// TwinCAT 3 PLC project PLC1
// ProgramVersion: 3.1.4026.25
// libraries:
//   Tc2_EtherCAT, * (Beckhoff Automation GmbH)
//   Tc2_MC2, * (Beckhoff Automation GmbH)
//   Tc2_Standard, * (Beckhoff Automation GmbH)
//   Tc2_System, * (Beckhoff Automation GmbH)
// project tree:
//   DUTs/ ST_DISDiagnosisMX.TcDUT, ST_DISInputsMX.TcDUT, ST_DOSDiagnosisMX.TcDUT, ST_DOSOutputsMX.TcDUT, ST_EFUInputsMX.TcDUT, ST_EFUOutputsMX.TcDUT, ST_IoModulMO1008.TcDUT, ST_IoModulMO2008.TcDUT, ST_IoModulMO2338.TcDUT, ST_MS4208.TcDUT, ST_PSUInputsMX.TcDUT
//   / PlcTask.TcTTO
//   POUs/ FB_RunOutputs.TcPOU, MAIN.TcPOU
// real-time tasks:
//   TASK PlcTask: cycle T#10ms, priority 20, ADS port 350
// motion (NC):
//   TASK NC-Task 1 SAF: cycle T#2ms, priority 4, ADS port 501
//   TASK NC-Task 1 SVB: cycle T#10ms, priority 8, ADS port 511
//   AXIS Axis 1 (id 1)
//     Dynamic: Acceleration=547.653, Deceleration=547.653, Jerk=1642.959
//     Velo: RefSearch=3.65102, RefSync=3.65102, SlowManual=12.5, FastManual=75, Fast=365.102, Maximum=365.102
//     OtherSettings: AllowMotionCmdToSlave=true
//     encoder EncType=19
//       EncPara: ScaleFactorNumerator=5, ScaleFactorDenominator=1048576, MaxCount=#xffffffff
//     drive DrvType=16
//       DrvPara: MaxCount=#xffffffff, DriveControlDWord=#x00020100
//         Analog: VeloReferenz=401.6122, VeloScale=32, TorqueSetpointScale=10, ScaleFactorActTorque=0.1
//         TimeComp: TaskDelayCycles=1
//     controller CtrType=1
//       CtrPara: PriorControlFactor=1
//         Observer: BandWidth=20
// I/O:
//   DEVICE Device 1 (EtherCAT), AmsNetId 192.168.7.189.2.1
//     Term 1 (MB1200-0000) [MB1200-0000 MX EtherCAT infeed]
//       Term 2 (MB1100-0002) [MB1100-0002 (Bluetooth gateway)]
//         Term 3 (MX Occupied Slot) [MX occupied Slot]
//         Term 4 (MX Occupied Slot) [MX occupied Slot]
//         Term 5 (MX Occupied Slot) [MX occupied Slot]
//         Term 6 (MS1010-1002-1334) [MS1010-1002-1334 Power infeed + forwarding, 230 V AC/10 A, 24 V DC/7A power supply, B17]
//         Term 7 (MO7221-0000-1114) [MO7221-0000-1114 1-channel motion interface, servomotor, 24 V DC/8 A, OCT, B17]
//           startup 32785:21 := 0E01 // DRV Motor Settings Ch.1 / Commutation offset
//           startup 32785:27 := E02E0000 // DRV Motor Settings Ch.1 / Motor speed limitation
//           startup 28688:3 := 08 // DRV Outputs Ch.1 / Modes of operation
//           startup 28688:16 := FF7F // DRV Outputs Ch.1 / Positive torque limit value
//           startup 28688:17 := FF7F // DRV Outputs Ch.1 / Negative torque limit value
//           startup 32784:87 := 64 // DRV Amplifier Settings Ch.1 / Position loop velocity feed forward gain
//           startup 32784:109 := 64000000 // DRV Amplifier Settings Ch.1 / Torque feed forward gain
//           startup 28688:11 := D007 // DRV Outputs Ch.1 / Torque limitation
//           startup 32784:19 := 9B00 // DRV Amplifier Settings Ch.1 / Current loop proportional gain
//           startup 32784:18 := 1200 // DRV Amplifier Settings Ch.1 / Current loop integral time
//           startup 32784:21 := C5000000 // DRV Amplifier Settings Ch.1 / Velocity loop proportional gain
//           startup 32784:20 := 96000000 // DRV Amplifier Settings Ch.1 / Velocity loop integral time
//         Term 8 (MB1120-0000) [MB1120 backplane junction]
//           Term 9 (MS4208-2003-1112) [MS4208-2003-1112 EtherCAT power output, EtherCAT, 24 V DC, 8 A, M12, switchable]
//             Term 24 (EK1100) [EK1100 EtherCAT Coupler (2A E-Bus)]
//               Term 25 (ED1008) [ED1008 | 8-ch. dig. input, 24 V DC, 3 ms, push-in]
//               Term 26 (ED2008) [ED2008 | 8-ch. dig. output, 24 V DC, 0.5 A, push-in]
//               Term 31 (ED4078) [ED4078 | 8-ch. ana. output, multi-function, ±10 V, ±20 mA, 16 bit, single-ended, 2 ksps, push-in]
//               Term 27 (ED5112) [ED5112 | 2-ch. encoder interface, incremental, 5 V DC (DIFF RS422, TTL, open collector), 5 MHz, push-in, 2 x AB/1 x ABC]
//               Term 32 (EL9011) [EL9011 End Terminal]
//         Term 10 (MO1008-0000-1111) [MO1008-0000-1111 8 Ch. Dig. Input 24V, M8]
//         Term 11 (MO2008-0000-1111) [MO2008-0000-1111 8 Ch. Dig. Output 24V, M8]
//         Term 12 (MO2338-0000-1112) [MO2338-0000-1112 8 Ch. digital combi 24V 0.5A, M12]
//         Term 15 (EL9011) [EL9011 End Terminal]
//       Term 13 (MS1110-0000) [MS1110-0000 | System module, EtherCAT extension]
// variable links:
//   NC-Task 1 SAF/Axes/Axis 1 <-> Device 1 (EtherCAT)/Term 1 (MB1200-0000)/Term 2 (MB1100-0002)/Term 7 (MO7221-0000-1114)
//     Drive/Inputs/In/nDataIn1 <-> DRV Following error actual value/Following error actual value
//     Drive/Inputs/In/nDataIn3[0] <-> DRV Torque actual value/Torque actual value
//     Drive/Inputs/In/nDcOutputTime <-> InfoData/DcOutputShift
//     Drive/Inputs/In/nState1 <-> DRV Statusword/Statusword
//     Drive/Inputs/In/nState2 <-> DRV Statusword/Statusword @bit 8
//     Drive/Inputs/In/nState4 @bit 1 <-> WcState/InputToggle
//     Drive/Inputs/In/nState4 <-> WcState/WcState
//     Drive/Outputs/Out/nCtrl1 <-> DRV Controlword/Controlword
//     Drive/Outputs/Out/nCtrl2 <-> DRV Controlword/Controlword @bit 8
//     Drive/Outputs/Out/nDataOut1 <-> DRV Target position/Target position
//     Enc/Inputs/In/nDataIn1 <-> FB Position/Position
//     Enc/Inputs/In/nDcInputTime <-> InfoData/DcInputShift
//     Enc/Inputs/In/nState4 @bit 1 <-> WcState/InputToggle
//     Enc/Inputs/In/nState4 <-> WcState/WcState
//   PLC1/PLC1 Instance <-> Device 1 (EtherCAT)
//     PlcTask Inputs/MAIN.nConfiguredSlaveCount <-> InfoData/CfgSlaveCount
//     PlcTask Inputs/MAIN.stAMSNetID <-> InfoData/AmsNetId
//   PLC1/PLC1 Instance <-> Device 1 (EtherCAT)/Term 1 (MB1200-0000)/Term 2 (MB1100-0002)
//     PlcTask Outputs/MAIN.bActivatePairingMode <-> BTG Outputs/Control/Activate Pairing
//     PlcTask Outputs/MAIN.bEnableBluetoothDiagnosis <-> BTG Outputs/Control/Enable Bluetooth
//   PLC1/PLC1 Instance <-> Device 1 (EtherCAT)/Term 1 (MB1200-0000)/Term 2 (MB1100-0002)/Term 10 (MO1008-0000-1111)
//     PlcTask Inputs/MAIN.stIoModulSlot8.stDISDiagnosis.bWirebreakCh1 <-> DIP Diagnosis/Wirebreak Ch1 X01-4
//     PlcTask Inputs/MAIN.stIoModulSlot8.stDISDiagnosis.bWirebreakCh2 <-> DIP Diagnosis/Wirebreak Ch2 X02-4
//     PlcTask Inputs/MAIN.stIoModulSlot8.stDISDiagnosis.bWirebreakCh3 <-> DIP Diagnosis/Wirebreak Ch3 X03-4
//     PlcTask Inputs/MAIN.stIoModulSlot8.stDISDiagnosis.bWirebreakCh4 <-> DIP Diagnosis/Wirebreak Ch4 X04-4
//     PlcTask Inputs/MAIN.stIoModulSlot8.stDISDiagnosis.bWirebreakCh5 <-> DIP Diagnosis/Wirebreak Ch5 X05-4
//     PlcTask Inputs/MAIN.stIoModulSlot8.stDISDiagnosis.bWirebreakCh6 <-> DIP Diagnosis/Wirebreak Ch6 X06-4
//     PlcTask Inputs/MAIN.stIoModulSlot8.stDISDiagnosis.bWirebreakCh7 <-> DIP Diagnosis/Wirebreak Ch7 X07-4
//     PlcTask Inputs/MAIN.stIoModulSlot8.stDISDiagnosis.bWirebreakCh8 <-> DIP Diagnosis/Wirebreak Ch8 X08-4
//     PlcTask Inputs/MAIN.stIoModulSlot8.stDISInputs.bInputCh1 <-> DIP Input/Input Ch1 X01-4
//     PlcTask Inputs/MAIN.stIoModulSlot8.stDISInputs.bInputCh2 <-> DIP Input/Input Ch2 X02-4
//     PlcTask Inputs/MAIN.stIoModulSlot8.stDISInputs.bInputCh3 <-> DIP Input/Input Ch3 X03-4
//     PlcTask Inputs/MAIN.stIoModulSlot8.stDISInputs.bInputCh4 <-> DIP Input/Input Ch4 X04-4
//     PlcTask Inputs/MAIN.stIoModulSlot8.stDISInputs.bInputCh5 <-> DIP Input/Input Ch5 X05-4
//     PlcTask Inputs/MAIN.stIoModulSlot8.stDISInputs.bInputCh6 <-> DIP Input/Input Ch6 X06-4
//     PlcTask Inputs/MAIN.stIoModulSlot8.stDISInputs.bInputCh7 <-> DIP Input/Input Ch7 X07-4
//     PlcTask Inputs/MAIN.stIoModulSlot8.stDISInputs.bInputCh8 <-> DIP Input/Input Ch8 X08-4
//     PlcTask Inputs/MAIN.stIoModulSlot8.stEFUInputs.bEnabled <-> EFU Inputs/Enabled
//     PlcTask Inputs/MAIN.stIoModulSlot8.stEFUInputs.bError <-> EFU Inputs/Error
//     PlcTask Inputs/MAIN.stIoModulSlot8.stEFUInputs.bTripped <-> EFU Inputs/Tripped
//     PlcTask Inputs/MAIN.stIoModulSlot8.stEFUInputs.bWarning <-> EFU Inputs/Warning
//     PlcTask Inputs/MAIN.stIoModulSlot8.stEFUInputs.fCurrent <-> EFU Inputs/Current
//     PlcTask Outputs/MAIN.stIoModulSlot8.stEFUOutputs.ControlViaProcessData <-> EFU Outputs/Control Via Process Data
//     PlcTask Outputs/MAIN.stIoModulSlot8.stEFUOutputs.bEnable <-> EFU Outputs/Enable
//     PlcTask Outputs/MAIN.stIoModulSlot8.stEFUOutputs.bReset <-> EFU Outputs/Reset
//   PLC1/PLC1 Instance <-> Device 1 (EtherCAT)/Term 1 (MB1200-0000)/Term 2 (MB1100-0002)/Term 11 (MO2008-0000-1111)
//     PlcTask Inputs/MAIN.stIoModulSlot9.stDOSDiagnosis.bOpenLoadCh1 <-> DOS Diagnosis/Open load Ch1 X01-4
//     PlcTask Inputs/MAIN.stIoModulSlot9.stDOSDiagnosis.bOpenLoadCh2 <-> DOS Diagnosis/Open load Ch2 X02-4
//     PlcTask Inputs/MAIN.stIoModulSlot9.stDOSDiagnosis.bOpenLoadCh3 <-> DOS Diagnosis/Open load Ch3 X03-4
//     PlcTask Inputs/MAIN.stIoModulSlot9.stDOSDiagnosis.bOpenLoadCh4 <-> DOS Diagnosis/Open load Ch4 X04-4
//     PlcTask Inputs/MAIN.stIoModulSlot9.stDOSDiagnosis.bOpenLoadCh5 <-> DOS Diagnosis/Open load Ch5 X05-4
//     PlcTask Inputs/MAIN.stIoModulSlot9.stDOSDiagnosis.bOpenLoadCh6 <-> DOS Diagnosis/Open load Ch6 X06-4
//     PlcTask Inputs/MAIN.stIoModulSlot9.stDOSDiagnosis.bOpenLoadCh7 <-> DOS Diagnosis/Open load Ch7 X07-4
//     PlcTask Inputs/MAIN.stIoModulSlot9.stDOSDiagnosis.bOpenLoadCh8 <-> DOS Diagnosis/Open load Ch8 X08-4
//     PlcTask Inputs/MAIN.stIoModulSlot9.stDOSDiagnosis.bOvercurrentCh1 <-> DOS Diagnosis/Overcurrent Ch1 X01-4
//     PlcTask Inputs/MAIN.stIoModulSlot9.stDOSDiagnosis.bOvercurrentCh2 <-> DOS Diagnosis/Overcurrent Ch2 X02-4
//     PlcTask Inputs/MAIN.stIoModulSlot9.stDOSDiagnosis.bOvercurrentCh3 <-> DOS Diagnosis/Overcurrent Ch3 X03-4
//     PlcTask Inputs/MAIN.stIoModulSlot9.stDOSDiagnosis.bOvercurrentCh4 <-> DOS Diagnosis/Overcurrent Ch4 X04-4
//     PlcTask Inputs/MAIN.stIoModulSlot9.stDOSDiagnosis.bOvercurrentCh5 <-> DOS Diagnosis/Overcurrent Ch5 X05-4
//     PlcTask Inputs/MAIN.stIoModulSlot9.stDOSDiagnosis.bOvercurrentCh6 <-> DOS Diagnosis/Overcurrent Ch6 X06-4
//     PlcTask Inputs/MAIN.stIoModulSlot9.stDOSDiagnosis.bOvercurrentCh7 <-> DOS Diagnosis/Overcurrent Ch7 X07-4
//     PlcTask Inputs/MAIN.stIoModulSlot9.stDOSDiagnosis.bOvercurrentCh8 <-> DOS Diagnosis/Overcurrent Ch8 X08-4
//     PlcTask Inputs/MAIN.stIoModulSlot9.stDOSDiagnosis.bOverloadCh1 <-> DOS Diagnosis/Overload Ch1 X01-4
//     PlcTask Inputs/MAIN.stIoModulSlot9.stDOSDiagnosis.bOverloadCh2 <-> DOS Diagnosis/Overload Ch2 X02-4
//     PlcTask Inputs/MAIN.stIoModulSlot9.stDOSDiagnosis.bOverloadCh3 <-> DOS Diagnosis/Overload Ch3 X03-4
//     PlcTask Inputs/MAIN.stIoModulSlot9.stDOSDiagnosis.bOverloadCh4 <-> DOS Diagnosis/Overload Ch4 X04-4
//     PlcTask Inputs/MAIN.stIoModulSlot9.stDOSDiagnosis.bOverloadCh5 <-> DOS Diagnosis/Overload Ch5 X05-4
//     PlcTask Inputs/MAIN.stIoModulSlot9.stDOSDiagnosis.bOverloadCh6 <-> DOS Diagnosis/Overload Ch6 X06-4
//     PlcTask Inputs/MAIN.stIoModulSlot9.stDOSDiagnosis.bOverloadCh7 <-> DOS Diagnosis/Overload Ch7 X07-4
//     PlcTask Inputs/MAIN.stIoModulSlot9.stDOSDiagnosis.bOverloadCh8 <-> DOS Diagnosis/Overload Ch8 X08-4
//     PlcTask Inputs/MAIN.stIoModulSlot9.stDOSDiagnosis.bShortTo24VCh1 <-> DOS Diagnosis/Short to 24V Ch1 X01-4
//     PlcTask Inputs/MAIN.stIoModulSlot9.stDOSDiagnosis.bShortTo24VCh2 <-> DOS Diagnosis/Short to 24V Ch2 X02-4
//     PlcTask Inputs/MAIN.stIoModulSlot9.stDOSDiagnosis.bShortTo24VCh3 <-> DOS Diagnosis/Short to 24V Ch3 X03-4
//     PlcTask Inputs/MAIN.stIoModulSlot9.stDOSDiagnosis.bShortTo24VCh4 <-> DOS Diagnosis/Short to 24V Ch4 X04-4
//     PlcTask Inputs/MAIN.stIoModulSlot9.stDOSDiagnosis.bShortTo24VCh5 <-> DOS Diagnosis/Short to 24V Ch5 X05-4
//     PlcTask Inputs/MAIN.stIoModulSlot9.stDOSDiagnosis.bShortTo24VCh6 <-> DOS Diagnosis/Short to 24V Ch6 X06-4
//     PlcTask Inputs/MAIN.stIoModulSlot9.stDOSDiagnosis.bShortTo24VCh7 <-> DOS Diagnosis/Short to 24V Ch7 X07-4
//     PlcTask Inputs/MAIN.stIoModulSlot9.stDOSDiagnosis.bShortTo24VCh8 <-> DOS Diagnosis/Short to 24V Ch8 X08-4
//     PlcTask Inputs/MAIN.stIoModulSlot9.stEFUInputs.bEnabled <-> EFU Inputs/Enabled
//     PlcTask Inputs/MAIN.stIoModulSlot9.stEFUInputs.bError <-> EFU Inputs/Error
//     PlcTask Inputs/MAIN.stIoModulSlot9.stEFUInputs.bTripped <-> EFU Inputs/Tripped
//     PlcTask Inputs/MAIN.stIoModulSlot9.stEFUInputs.bWarning <-> EFU Inputs/Warning
//     PlcTask Inputs/MAIN.stIoModulSlot9.stEFUInputs.fCurrent <-> EFU Inputs/Current
//     PlcTask Outputs/MAIN.stIoModulSlot9.stDOSOutputs.bOutputCh1 <-> DOS Output/Output Ch1 X01-4
//     PlcTask Outputs/MAIN.stIoModulSlot9.stDOSOutputs.bOutputCh2 <-> DOS Output/Output Ch2 X02-4
//     PlcTask Outputs/MAIN.stIoModulSlot9.stDOSOutputs.bOutputCh3 <-> DOS Output/Output Ch3 X03-4
//     PlcTask Outputs/MAIN.stIoModulSlot9.stDOSOutputs.bOutputCh4 <-> DOS Output/Output Ch4 X04-4
//     PlcTask Outputs/MAIN.stIoModulSlot9.stDOSOutputs.bOutputCh5 <-> DOS Output/Output Ch5 X05-4
//     PlcTask Outputs/MAIN.stIoModulSlot9.stDOSOutputs.bOutputCh6 <-> DOS Output/Output Ch6 X06-4
//     PlcTask Outputs/MAIN.stIoModulSlot9.stDOSOutputs.bOutputCh7 <-> DOS Output/Output Ch7 X07-4
//     PlcTask Outputs/MAIN.stIoModulSlot9.stDOSOutputs.bOutputCh8 <-> DOS Output/Output Ch8 X08-4
//     PlcTask Outputs/MAIN.stIoModulSlot9.stEFUOutputs.ControlViaProcessData <-> EFU Outputs/Control Via Process Data
//     PlcTask Outputs/MAIN.stIoModulSlot9.stEFUOutputs.bEnable <-> EFU Outputs/Enable
//     PlcTask Outputs/MAIN.stIoModulSlot9.stEFUOutputs.bReset <-> EFU Outputs/Reset
//   PLC1/PLC1 Instance <-> Device 1 (EtherCAT)/Term 1 (MB1200-0000)/Term 2 (MB1100-0002)/Term 12 (MO2338-0000-1112)
//     PlcTask Inputs/MAIN.stIoModulSlot10.stDISDiagnosis.bWirebreakCh1 <-> DIP Diagnosis/Wirebreak Ch1 X01-4
//     PlcTask Inputs/MAIN.stIoModulSlot10.stDISDiagnosis.bWirebreakCh2 <-> DIP Diagnosis/Wirebreak Ch2 X01-2
//     PlcTask Inputs/MAIN.stIoModulSlot10.stDISDiagnosis.bWirebreakCh3 <-> DIP Diagnosis/Wirebreak Ch3 X02-4
//     PlcTask Inputs/MAIN.stIoModulSlot10.stDISDiagnosis.bWirebreakCh4 <-> DIP Diagnosis/Wirebreak Ch4 X02-2
//     PlcTask Inputs/MAIN.stIoModulSlot10.stDISDiagnosis.bWirebreakCh5 <-> DIP Diagnosis/Wirebreak Ch5 X03-4
//     PlcTask Inputs/MAIN.stIoModulSlot10.stDISDiagnosis.bWirebreakCh6 <-> DIP Diagnosis/Wirebreak Ch6 X03-2
//     PlcTask Inputs/MAIN.stIoModulSlot10.stDISDiagnosis.bWirebreakCh7 <-> DIP Diagnosis/Wirebreak Ch7 X04-4
//     PlcTask Inputs/MAIN.stIoModulSlot10.stDISDiagnosis.bWirebreakCh8 <-> DIP Diagnosis/Wirebreak Ch8 X04-2
//     PlcTask Inputs/MAIN.stIoModulSlot10.stDISInputs.bInputCh1 <-> DIP Input/Input Ch1 X01-4
//     PlcTask Inputs/MAIN.stIoModulSlot10.stDISInputs.bInputCh2 <-> DIP Input/Input Ch2 X01-2
//     PlcTask Inputs/MAIN.stIoModulSlot10.stDISInputs.bInputCh3 <-> DIP Input/Input Ch3 X02-4
//     PlcTask Inputs/MAIN.stIoModulSlot10.stDISInputs.bInputCh4 <-> DIP Input/Input Ch4 X02-2
//     PlcTask Inputs/MAIN.stIoModulSlot10.stDISInputs.bInputCh5 <-> DIP Input/Input Ch5 X03-4
//     PlcTask Inputs/MAIN.stIoModulSlot10.stDISInputs.bInputCh6 <-> DIP Input/Input Ch6 X03-2
//     PlcTask Inputs/MAIN.stIoModulSlot10.stDISInputs.bInputCh7 <-> DIP Input/Input Ch7 X04-4
//     PlcTask Inputs/MAIN.stIoModulSlot10.stDISInputs.bInputCh8 <-> DIP Input/Input Ch8 X04-2
//     PlcTask Inputs/MAIN.stIoModulSlot10.stDOSDiagnosis.bOvercurrentCh1 <-> DOS Diagnosis/Overcurrent Ch1 X01-4
//     PlcTask Inputs/MAIN.stIoModulSlot10.stDOSDiagnosis.bOvercurrentCh2 <-> DOS Diagnosis/Overcurrent Ch2 X01-2
//     PlcTask Inputs/MAIN.stIoModulSlot10.stDOSDiagnosis.bOvercurrentCh3 <-> DOS Diagnosis/Overcurrent Ch3 X02-4
//     PlcTask Inputs/MAIN.stIoModulSlot10.stDOSDiagnosis.bOvercurrentCh4 <-> DOS Diagnosis/Overcurrent Ch4 X02-2
//     PlcTask Inputs/MAIN.stIoModulSlot10.stDOSDiagnosis.bOvercurrentCh5 <-> DOS Diagnosis/Overcurrent Ch5 X03-4
//     PlcTask Inputs/MAIN.stIoModulSlot10.stDOSDiagnosis.bOvercurrentCh6 <-> DOS Diagnosis/Overcurrent Ch6 X03-2
//     PlcTask Inputs/MAIN.stIoModulSlot10.stDOSDiagnosis.bOvercurrentCh7 <-> DOS Diagnosis/Overcurrent Ch7 X04-4
//     PlcTask Inputs/MAIN.stIoModulSlot10.stDOSDiagnosis.bOvercurrentCh8 <-> DOS Diagnosis/Overcurrent Ch8 X04-2
//     PlcTask Inputs/MAIN.stIoModulSlot10.stDOSDiagnosis.bOverloadCh1 <-> DOS Diagnosis/Overload Ch1 X01-4
//     PlcTask Inputs/MAIN.stIoModulSlot10.stDOSDiagnosis.bOverloadCh2 <-> DOS Diagnosis/Overload Ch2 X01-2
//     PlcTask Inputs/MAIN.stIoModulSlot10.stDOSDiagnosis.bOverloadCh3 <-> DOS Diagnosis/Overload Ch3 X02-4
//     PlcTask Inputs/MAIN.stIoModulSlot10.stDOSDiagnosis.bOverloadCh4 <-> DOS Diagnosis/Overload Ch4 X02-2
//     PlcTask Inputs/MAIN.stIoModulSlot10.stDOSDiagnosis.bOverloadCh5 <-> DOS Diagnosis/Overload Ch5 X03-4
//     PlcTask Inputs/MAIN.stIoModulSlot10.stDOSDiagnosis.bOverloadCh6 <-> DOS Diagnosis/Overload Ch6 X03-2
//     PlcTask Inputs/MAIN.stIoModulSlot10.stDOSDiagnosis.bOverloadCh7 <-> DOS Diagnosis/Overload Ch7 X04-4
//     PlcTask Inputs/MAIN.stIoModulSlot10.stDOSDiagnosis.bOverloadCh8 <-> DOS Diagnosis/Overload Ch8 X04-2
//     PlcTask Inputs/MAIN.stIoModulSlot10.stDOSDiagnosis.bShortTo24VCh1 <-> DOS Diagnosis/Short to 24V Ch1 X01-4
//     PlcTask Inputs/MAIN.stIoModulSlot10.stDOSDiagnosis.bShortTo24VCh2 <-> DOS Diagnosis/Short to 24V Ch2 X01-2
//     PlcTask Inputs/MAIN.stIoModulSlot10.stDOSDiagnosis.bShortTo24VCh3 <-> DOS Diagnosis/Short to 24V Ch3 X02-4
//     PlcTask Inputs/MAIN.stIoModulSlot10.stDOSDiagnosis.bShortTo24VCh4 <-> DOS Diagnosis/Short to 24V Ch4 X02-2
//     PlcTask Inputs/MAIN.stIoModulSlot10.stDOSDiagnosis.bShortTo24VCh5 <-> DOS Diagnosis/Short to 24V Ch5 X03-4
//     PlcTask Inputs/MAIN.stIoModulSlot10.stDOSDiagnosis.bShortTo24VCh6 <-> DOS Diagnosis/Short to 24V Ch6 X03-2
//     PlcTask Inputs/MAIN.stIoModulSlot10.stDOSDiagnosis.bShortTo24VCh7 <-> DOS Diagnosis/Short to 24V Ch7 X04-4
//     PlcTask Inputs/MAIN.stIoModulSlot10.stDOSDiagnosis.bShortTo24VCh8 <-> DOS Diagnosis/Short to 24V Ch8 X04-2
//     PlcTask Inputs/MAIN.stIoModulSlot10.stEFUInputs.bEnabled <-> EFU Inputs/Enabled
//     PlcTask Inputs/MAIN.stIoModulSlot10.stEFUInputs.bError <-> EFU Inputs/Error
//     PlcTask Inputs/MAIN.stIoModulSlot10.stEFUInputs.bTripped <-> EFU Inputs/Tripped
//     PlcTask Inputs/MAIN.stIoModulSlot10.stEFUInputs.bWarning <-> EFU Inputs/Warning
//     PlcTask Inputs/MAIN.stIoModulSlot10.stEFUInputs.fCurrent <-> EFU Inputs/Current
//     PlcTask Outputs/MAIN.stIoModulSlot10.stDOSOutputs.bOutputCh1 <-> DOS Output/Output Ch1 X01-4
//     PlcTask Outputs/MAIN.stIoModulSlot10.stDOSOutputs.bOutputCh2 <-> DOS Output/Output Ch2 X01-2
//     PlcTask Outputs/MAIN.stIoModulSlot10.stDOSOutputs.bOutputCh3 <-> DOS Output/Output Ch3 X02-4
//     PlcTask Outputs/MAIN.stIoModulSlot10.stDOSOutputs.bOutputCh4 <-> DOS Output/Output Ch4 X02-2
//     PlcTask Outputs/MAIN.stIoModulSlot10.stDOSOutputs.bOutputCh5 <-> DOS Output/Output Ch5 X03-4
//     PlcTask Outputs/MAIN.stIoModulSlot10.stDOSOutputs.bOutputCh6 <-> DOS Output/Output Ch6 X03-2
//     PlcTask Outputs/MAIN.stIoModulSlot10.stDOSOutputs.bOutputCh7 <-> DOS Output/Output Ch7 X04-4
//     PlcTask Outputs/MAIN.stIoModulSlot10.stDOSOutputs.bOutputCh8 <-> DOS Output/Output Ch8 X04-2
//     PlcTask Outputs/MAIN.stIoModulSlot10.stEFUOutputs.ControlViaProcessData <-> EFU Outputs/Control Via Process Data
//     PlcTask Outputs/MAIN.stIoModulSlot10.stEFUOutputs.bEnable <-> EFU Outputs/Enable
//     PlcTask Outputs/MAIN.stIoModulSlot10.stEFUOutputs.bReset <-> EFU Outputs/Reset
//   PLC1/PLC1 Instance <-> Device 1 (EtherCAT)/Term 1 (MB1200-0000)/Term 2 (MB1100-0002)/Term 6 (MS1010-1002-1334)
//     PlcTask Inputs/MAIN.stPSUSlot3.bError <-> PSU Inputs/Error
//     PlcTask Inputs/MAIN.stPSUSlot3.bI2TWarning <-> PSU Inputs/I2T Warning
//     PlcTask Inputs/MAIN.stPSUSlot3.bWarning <-> PSU Inputs/Warning
//     PlcTask Inputs/MAIN.stPSUSlot3.fActualOutputCurrent <-> PSU Inputs/Output Current
//     PlcTask Inputs/MAIN.stPSUSlot3.fActualOutputVoltage <-> PSU Inputs/Output Voltage
//     PlcTask Inputs/MAIN.stPSUSlot3.nActualI2TUtilization <-> PSU Inputs/I2T Utilization
//     PlcTask Inputs/MAIN.stPSUSlot3.nInfoData1 <-> PSU Inputs/Info Data 1
//     PlcTask Inputs/MAIN.stPSUSlot3.nInfoData2 <-> PSU Inputs/Info Data 2
//   PLC1/PLC1 Instance <-> Device 1 (EtherCAT)/Term 1 (MB1200-0000)/Term 2 (MB1100-0002)/Term 8 (MB1120-0000)/Term 9 (MS4208-2003-1112)
//     PlcTask Inputs/MAIN.stMS4208Slot7.stEFUInputsUp1.bEnabled <-> EFU Up1 Inputs/Enabled
//     PlcTask Inputs/MAIN.stMS4208Slot7.stEFUInputsUp2.bEnabled <-> EFU Up2 Inputs/Enabled
//     PlcTask Inputs/MAIN.stMS4208Slot7.stEFUInputsUp1.bError <-> EFU Up1 Inputs/Error
//     PlcTask Inputs/MAIN.stMS4208Slot7.stEFUInputsUp2.bError <-> EFU Up2 Inputs/Error
//     PlcTask Inputs/MAIN.stMS4208Slot7.stEFUInputsUp1.bTripped <-> EFU Up1 Inputs/Tripped
//     PlcTask Inputs/MAIN.stMS4208Slot7.stEFUInputsUp2.bTripped <-> EFU Up2 Inputs/Tripped
//     PlcTask Inputs/MAIN.stMS4208Slot7.stEFUInputsUp1.bWarning <-> EFU Up1 Inputs/Warning
//     PlcTask Inputs/MAIN.stMS4208Slot7.stEFUInputsUp2.bWarning <-> EFU Up2 Inputs/Warning
//     PlcTask Inputs/MAIN.stMS4208Slot7.stEFUInputsUp1.fCurrent <-> EFU Up1 Inputs/Current
//     PlcTask Inputs/MAIN.stMS4208Slot7.stEFUInputsUp2.fCurrent <-> EFU Up2 Inputs/Current
//     PlcTask Inputs/MAIN.stMS4208Slot7.stEFUInputsUs.bEnabled <-> EFU Us Inputs/Enabled
//     PlcTask Inputs/MAIN.stMS4208Slot7.stEFUInputsUs.bError <-> EFU Us Inputs/Error
//     PlcTask Inputs/MAIN.stMS4208Slot7.stEFUInputsUs.bTripped <-> EFU Us Inputs/Tripped
//     PlcTask Inputs/MAIN.stMS4208Slot7.stEFUInputsUs.bWarning <-> EFU Us Inputs/Warning
//     PlcTask Inputs/MAIN.stMS4208Slot7.stEFUInputsUs.fCurrent <-> EFU Us Inputs/Current
//     PlcTask Outputs/MAIN.stMS4208Slot7.stEFUOutputsUp1.ControlViaProcessData <-> EFU Up1 Outputs/Control via Process Data
//     PlcTask Outputs/MAIN.stMS4208Slot7.stEFUOutputsUp2.ControlViaProcessData <-> EFU Up2 Outputs/Control via Process Data
//     PlcTask Outputs/MAIN.stMS4208Slot7.stEFUOutputsUp1.bEnable <-> EFU Up1 Outputs/Enable
//     PlcTask Outputs/MAIN.stMS4208Slot7.stEFUOutputsUp2.bEnable <-> EFU Up2 Outputs/Enable
//     PlcTask Outputs/MAIN.stMS4208Slot7.stEFUOutputsUp1.bReset <-> EFU Up1 Outputs/Reset
//     PlcTask Outputs/MAIN.stMS4208Slot7.stEFUOutputsUp2.bReset <-> EFU Up2 Outputs/Reset
//     PlcTask Outputs/MAIN.stMS4208Slot7.stEFUOutputsUs.ControlViaProcessData <-> EFU Us Outputs/Control via Process Data
//     PlcTask Outputs/MAIN.stMS4208Slot7.stEFUOutputsUs.bEnable <-> EFU Us Outputs/Enable
//     PlcTask Outputs/MAIN.stMS4208Slot7.stEFUOutputsUs.bReset <-> EFU Us Outputs/Reset
//   PLC1/PLC1 Instance <-> NC-Task 1 SAF/Axes/Axis 1
//     PlcTask Inputs/MAIN.Axis1.NcToPlc <-> Outputs/ToPlc
//     PlcTask Outputs/MAIN.Axis1.PlcToNc <-> Inputs/FromPlc

CONFIGURATION PLC1
    RESOURCE PLC ON TwinCAT3
        TASK PlcTask(INTERVAL := T#10ms, PRIORITY := 20);
        PROGRAM MAIN WITH PlcTask : MAIN;
    END_RESOURCE
END_CONFIGURATION

// ---- DUTs/ST_DISDiagnosisMX.TcDUT
TYPE ST_DISDiagnosisMX :
STRUCT
	bWirebreakCh1 AT%I* : BOOL;
	bWirebreakCh2 AT%I* : BOOL;
	bWirebreakCh3 AT%I* : BOOL;
	bWirebreakCh4 AT%I* : BOOL;
	bWirebreakCh5 AT%I* : BOOL;
	bWirebreakCh6 AT%I* : BOOL;
	bWirebreakCh7 AT%I* : BOOL;
	bWirebreakCh8 AT%I* : BOOL;
END_STRUCT
END_TYPE

// ---- DUTs/ST_DISInputsMX.TcDUT
TYPE ST_DISInputsMX :
STRUCT
	bInputCh1 AT%I* : BOOL;
	bInputCh2 AT%I* : BOOL;
	bInputCh3 AT%I* : BOOL;
	bInputCh4 AT%I* : BOOL;
	bInputCh5 AT%I* : BOOL;
	bInputCh6 AT%I* : BOOL;
	bInputCh7 AT%I* : BOOL;
	bInputCh8 AT%I* : BOOL;
END_STRUCT
END_TYPE

// ---- DUTs/ST_DOSDiagnosisMX.TcDUT
TYPE ST_DOSDiagnosisMX :
STRUCT
	bOvercurrentCh1 	AT%I*	: BOOL;
	bOverloadCh1		AT%I*	: BOOL;
	bOpenLoadCh1 		AT%I*	: BOOL;
	bShortTo24VCh1 		AT%I*	: BOOL;
	bOvercurrentCh2 	AT%I*	: BOOL;
	bOverloadCh2		AT%I*	: BOOL;
	bOpenLoadCh2 		AT%I*	: BOOL;
	bShortTo24VCh2 		AT%I*	: BOOL;
	bOvercurrentCh3 	AT%I*	: BOOL;
	bOverloadCh3		AT%I*	: BOOL;
	bOpenLoadCh3 		AT%I*	: BOOL;
	bShortTo24VCh3 		AT%I*	: BOOL;
	bOvercurrentCh4 	AT%I*	: BOOL;
	bOverloadCh4		AT%I*	: BOOL;
	bOpenLoadCh4 		AT%I*	: BOOL;
	bShortTo24VCh4 		AT%I*	: BOOL;
	bOvercurrentCh5 	AT%I*	: BOOL;
	bOverloadCh5		AT%I*	: BOOL;
	bOpenLoadCh5 		AT%I*	: BOOL;
	bShortTo24VCh5 		AT%I*	: BOOL;
	bOvercurrentCh6 	AT%I*	: BOOL;
	bOverloadCh6		AT%I*	: BOOL;
	bOpenLoadCh6 		AT%I*	: BOOL;
	bShortTo24VCh6 		AT%I*	: BOOL;
	bOvercurrentCh7 	AT%I*	: BOOL;
	bOverloadCh7		AT%I*	: BOOL;
	bOpenLoadCh7 		AT%I*	: BOOL;
	bShortTo24VCh7 		AT%I*	: BOOL;
	bOvercurrentCh8 	AT%I*	: BOOL;
	bOverloadCh8		AT%I*	: BOOL;
	bOpenLoadCh8 		AT%I*	: BOOL;
	bShortTo24VCh8 		AT%I*	: BOOL;
END_STRUCT
END_TYPE

// ---- DUTs/ST_DOSOutputsMX.TcDUT
TYPE ST_DOSOutputsMX :
STRUCT
	bOutputCh1	AT%Q*: BOOL;
	bOutputCh2	AT%Q*: BOOL;
	bOutputCh3	AT%Q*: BOOL;
	bOutputCh4	AT%Q*: BOOL;
	bOutputCh5	AT%Q*: BOOL;
	bOutputCh6	AT%Q*: BOOL;
	bOutputCh7	AT%Q*: BOOL;
	bOutputCh8	AT%Q*: BOOL;
END_STRUCT
END_TYPE

// ---- DUTs/ST_EFUInputsMX.TcDUT
TYPE ST_EFUInputsMX :
STRUCT
	bWarning 	AT%I*	: BOOL;
	bError 		AT%I*	: BOOL;
	bTripped 	AT%I*	: BOOL;
	bEnabled 	AT%I*	: BOOL;
	//InputCycleCounter : BYTE;
	fCurrent 	AT%I*	: REAL;
END_STRUCT
END_TYPE

// ---- DUTs/ST_EFUOutputsMX.TcDUT
TYPE ST_EFUOutputsMX :
STRUCT
	bEnable 				AT%Q*	: BOOL;
	ControlViaProcessData 	AT%Q*	: BOOL;
	bReset 					AT%Q*	: BOOL;
END_STRUCT
END_TYPE

// ---- DUTs/ST_IoModulMO1008.TcDUT
TYPE ST_IoModulMO1008 :
STRUCT
	stDISInputs : ST_DISInputsMX;
	stDISDiagnosis : ST_DISDiagnosisMX;
	stEFUInputs : ST_EFUInputsMX;
	stEFUOutputs : ST_EFUOutputsMX;
END_STRUCT
END_TYPE

// ---- DUTs/ST_IoModulMO2008.TcDUT
TYPE ST_IoModulMO2008 :
STRUCT
	stDOSOutputs : ST_DOSOutputsMX;
	stDOSDiagnosis : ST_DOSDiagnosisMX;
	stEFUInputs : ST_EFUInputsMX;
	stEFUOutputs : ST_EFUOutputsMX;
END_STRUCT
END_TYPE

// ---- DUTs/ST_IoModulMO2338.TcDUT
TYPE ST_IoModulMO2338 :
STRUCT
	stDISInputs : ST_DISInputsMX;
	stDOSOutputs : ST_DOSOutputsMX;
	stDISDiagnosis : ST_DISDiagnosisMX;
	stDOSDiagnosis : ST_DOSDiagnosisMX;
	stEFUInputs : ST_EFUInputsMX;
	stEFUOutputs : ST_EFUOutputsMX;
END_STRUCT
END_TYPE

// ---- DUTs/ST_MS4208.TcDUT
TYPE ST_MS4208 :
STRUCT
	stEFUInputsUs		:		ST_EFUInputsMX;
	stEFUInputsUp1		:		ST_EFUInputsMX;
	stEFUInputsUp2		:		ST_EFUInputsMX;
	stEFUOutputsUs		:		ST_EFUOutputsMX;
	stEFUOutputsUp1		:		ST_EFUOutputsMX;
	stEFUOutputsUp2		:		ST_EFUOutputsMX;
END_STRUCT
END_TYPE

// ---- DUTs/ST_PSUInputsMX.TcDUT
TYPE ST_PSUInputsMX :
STRUCT
	bWarning 				AT%I* : BOOL;
	bError 					AT%I* : BOOL;
	bI2TWarning 			AT%I* : BOOL;
	nInpuCycleCounter 		AT%I* : UINT;
	fActualOutputVoltage 	AT%I* : REAL;
	fActualOutputCurrent 	AT%I* : REAL;
	nActualI2TUtilization 	AT%I* : USINT;
	nInfoData1 				AT%I* : UINT;
	nInfoData2 				AT%I* : UINT;
END_STRUCT
END_TYPE

// ---- POUs/MAIN.TcPOU
PROGRAM MAIN
VAR
	stPSUSlot3		:	ST_PSUInputsMX;
	stMS4208Slot7	:	ST_MS4208;
	stIoModulSlot8	:	ST_IoModulMO1008;
	stIoModulSlot9	:	ST_IoModulMO2008;
	stIoModulSlot10	:	ST_IoModulMo2338;
	
	fTest			:	REAL := 3.141;
	
	bEnableBluetoothDiagnosis	AT%Q* 	:  	BOOL := TRUE;
	bActivatePairingMode		AT%Q*	:	BOOL := TRUE;
	
	fbRunOutputs						:	FB_RunOutputs;
	
	fbGetAllSlaveStates 				: FB_EcGetAllSlaveStates;
	fbGetAllSlaveConfigs				: FB_EcGetConfSlaves;
	stAMSNetID					AT %I*	: AMSNETID;
	arrEtherCATSlaves					: ARRAY [0..EC_MAX_SLAVES] OF ST_EcSlaveState;
	arrEtherCATSlavesConf				: ARRAY [0..EC_MAX_SLAVES] OF ST_EcSlaveConfigData;
	nConfiguredSlaveCount		AT %I*	: UINT;
	nFoundSlaveCount					: UINT;

	nEtherCATDiagState					: UDINT := 0;
	nForLoopIdx							: UINT := 0;
	bError: BOOL;
	fbRequestSlaveState: FB_EcReqSlaveState;
	
	nStackIDX							: UINT := 0;
	arrStack							: ARRAY [0..EC_MAX_SLAVES] OF UINT;
	
	Axis1  								: AXIS_REF;
	fbEnableAxis						: MC_Power;
	bEnableAxis							: BOOL;
	fbJog								: MC_Jog;
	bForwardJog: BOOL;
	bBackwardJog: BOOL;
	fbEnableHardwareButton: R_TRIG;
END_VAR

fbRunOutputs(bEnable:=TRUE , tStepSpeed:=T#500MS , tCycleDelay:=T#1000MS , Outputs_MX:=stIoModulSlot9.stDOSOutputs );
(* This should be a State Machine Doesn't have to be FAST*)
// Loop through configured number of slaves
// Capture which slaves are NOT in OP
// Clear Errors on List
// Set Devices to OP
fbGetAllSlaveStates(sNetId:= F_CreateAmsNetId(stAMSNetID), pStateBuf:=ADR(arrEtherCATSlaves), cbBufLen:=SIZEOF(arrEtherCATSlaves), nSlaves=>nFoundSlaveCount);
fbGetAllSlaveConfigs(sNetId:=F_CreateAmsNetId(stAMSNetID), pArrEcConfSlaveInfo:=ADR(arrEtherCATSlavesConf), cbBufLen:=SIZEOF(arrEtherCATSlavesConf));
fbRequestSlaveState(
	sNetId:=F_CreateAmsNetId(stAMSNetID) , 
	nSlaveAddr:= , 
	bExecute:= , 
	tTimeout:= , 
	state:= 8, 
	bBusy=> , 
	bError=> , 
	nErrId=> );

CASE nEtherCATDiagState OF
	0: //INIT
	fbGetAllSlaveConfigs.bExecute:=TRUE;
	nEtherCATDiagState:=nEtherCATDiagState+1;
	
	1: //SET READ
	fbGetAllSlaveStates.bExecute := TRUE;
	IF fbGetAllSlaveStates.bBusy THEN
		nEtherCATDiagState:=nEtherCATDiagState+1;
	END_IF
	
	2: //READ DONE
	IF NOT(fbGetAllSlaveStates.bBusy OR fbGetAllSlaveStates.bError) THEN
		nEtherCATDiagState:=nEtherCATDiagState+1;
		bError:=FALSE;
	ELSE
		nEtherCATDiagState:=999;
	END_IF
	
	3: //CHECK ERRORS
	FOR nForLoopIdx:=0 TO nFoundSlaveCount-1 BY 1 DO
		IF arrEtherCATSlaves[nForLoopIdx].deviceState <> 8 // Are we in OP
			AND arrEtherCATSlavesConf[nForLoopIdx].stSlaveIdentity.productCode<>90320  // Ignore MX0001 "EMPTY" modules 
		THEN
			arrStack[nStackIDX]:=nForLoopIdx;
			nStackIDX:=nStackIDX+1;
		END_IF
	END_FOR
	nEtherCATDiagState:=nEtherCATDiagState+1;
	
	4: //TRY SET OP
	IF nStackIDX>0 THEN
		fbRequestSlaveState.nSlaveAddr:=arrEtherCATSlavesConf[arrStack[0]].nAddr;
		fbRequestSlaveState.bExecute:=TRUE;
		nStackIDX:=nStackIDX-1;
		nEtherCATDiagState:=nEtherCATDiagState+1;
	ELSE
		nEtherCATDiagState:=6; // Start Over Actually
	END_IF
	
	5: //CHECK DONE
	IF NOT(fbRequestSlaveState.bBusy) THEN
		fbRequestSlaveState.bExecute:=FALSE;
		nEtherCATDiagState:=nEtherCATDiagState-1;
	END_IF
	
	6: //READ AGAIN
	fbGetAllSlaveStates.bExecute:=FALSE;
	nEtherCATDiagState:=1;
	
	999: //ERROR
	;
	
END_CASE

fbEnableHardwareButton(CLK:= stIoModulSlot10.stDISInputs.bInputCh4);
IF fbEnableHardwareButton.Q THEN
	IF bEnableAxis THEN
		bEnableAxis:=FALSE;
	ELSE
		bEnableAxis:=TRUE;
	END_IF
END_IF

Axis1.ReadStatus();
fbEnableAxis(
	Axis:=Axis1 , 
	Enable:=bEnableAxis , 
	Enable_Positive:=bEnableAxis , 
	Enable_Negative:=bEnableAxis , 
	Override:=100.0);
	
fbJog(
	Axis:=Axis1 , 
	JogForward:=bForwardJog OR stIoModulSlot10.stDISInputs.bInputCh2 , 
	JogBackwards:=bBackwardJog OR stIoModulSlot10.stDISInputs.bInputCh6 , 
	Mode:=MC_Aborting , 
	Velocity:=100.0 );
	
stIoModulSlot10.stDOSOutputs.bOutputCh3:=fbEnableAxis.Status;
stIoModulSlot10.stDOSOutputs.bOutputCh1:=fbJog.JogForward;
stIoModulSlot10.stDOSOutputs.bOutputCh5:=fbJog.JogForward;

IF _TaskInfo[1].FirstCycle THEN
	stMS4208Slot7.stEFUOutputsUp1.ControlViaProcessData:=TRUE;
	stMS4208Slot7.stEFUInputsUp1.bEnabled:=TRUE;
	stMS4208Slot7.stEFUOutputsUp2.ControlViaProcessData:=TRUE;
	stMS4208Slot7.stEFUInputsUp2.bEnabled:=TRUE;
	stMS4208Slot7.stEFUOutputsUs.ControlViaProcessData:=TRUE;
	stMS4208Slot7.stEFUInputsUs.bEnabled:=TRUE;
END_IF

END_PROGRAM

// ---- POUs/FB_RunOutputs.TcPOU
FUNCTION_BLOCK FB_RunOutputs
VAR_INPUT
	bEnable : BOOL;
	tStepSpeed : TIME;
	tCycleDelay : TIME;
END_VAR
VAR
	nStep: INT;
	fbStepTimer: TON;
	fbCycleDelay: TON;
	nShiftReg : BYTE;
END_VAR
VAR_IN_OUT
	Outputs_MX : ST_DOSOutputsMX;
END_VAR

CASE nStep OF
0:
	fbStepTimer.IN := FALSE;
	fbCycleDelay.IN := FALSE;
	IF bEnable THEN
		nShiftReg:=1;
		fbStepTimer.IN:=TRUE;
		nStep:=nStep+1;
	END_IF
	
1:
	IF fbStepTimer.Q THEN
		fbStepTimer.IN:=FALSE;
		nStep:=nStep+1;
	END_IF

2:
	nShiftReg:=SHL(nShiftReg,1);
	IF Outputs_MX.bOutputCh8 THEN
		fbCycleDelay.IN:=TRUE;
		nStep:=nStep+1;	
	ELSE
		fbStepTimer.IN:=TRUE;
		nStep:=nStep-1;
	END_IF

3:
	IF fbCycleDelay.Q THEN
		nShiftReg:=1;
		fbStepTimer.IN:=TRUE;
		fbCycleDelay.IN:=FALSE;
		nStep:=1;
	END_IF

999:
	nShiftReg:=0;
	fbCycleDelay.IN:=FALSE;
	fbStepTimer.IN:=FALSE;
	nStep:=0;

END_CASE
fbStepTimer(PT:=tStepSpeed);
fbCycleDelay(PT:=tCycleDelay);
IF NOT(bEnable) THEN
	nStep:=999;
END_IF
Outputs_MX.bOutputCh8:=nShiftReg.7;
Outputs_MX.bOutputCh7:=nShiftReg.6;
Outputs_MX.bOutputCh6:=nShiftReg.5;
Outputs_MX.bOutputCh5:=nShiftReg.4;
Outputs_MX.bOutputCh4:=nShiftReg.3;
Outputs_MX.bOutputCh3:=nShiftReg.2;
Outputs_MX.bOutputCh2:=nShiftReg.1;
Outputs_MX.bOutputCh1:=nShiftReg.0;

END_FUNCTION_BLOCK
